FUNCTION_BLOCK TwoConRingCTL (* Composite Function Block Type *)
  (* Standard: 61499-2 *)
  (* Version 0.2, 2003-12-05, JHC, Rockwell Automation, Renamed from NEWCOMPFB. *)
  (* Version 0.1, 2002-01-08, JHC, Rockwell Automation, Added DLY FB as example. *)
  (* Version 0.0, 2000-05-27, JHC, Rockwell Automation *)
  (* Compiler header: package fb.rt.cs725; *)
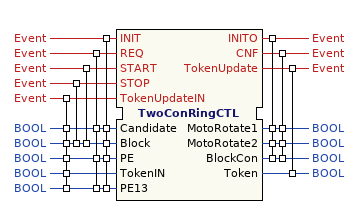
  EVENT_INPUT
    INIT WITH Candidate, Block, PE, PE13; (* Initialization Request *)
    REQ WITH Candidate, PE, PE13; (* Normal Execution Request *)
    START WITH Block;
    STOP WITH Block;
    TokenUpdateIN WITH Candidate, Block, PE, TokenIN, PE13;
  END_EVENT
  EVENT_OUTPUT
    INITO WITH MotoRotate1, MotoRotate2, BlockCon; (* Initialization Confirm *)
    CNF WITH MotoRotate1, MotoRotate2, BlockCon; (* Execution Confirmation *)
    TokenUpdate WITH Token;
  END_EVENT
  VAR_INPUT
    Candidate : BOOL;
    Block : BOOL;
    PE : BOOL;
    TokenIN : BOOL;
    PE13 : BOOL;
  END_VAR
  VAR_OUTPUT
    MotoRotate1 : BOOL;
    MotoRotate2 : BOOL;
    BlockCon : BOOL;
    Token : BOOL;
  END_VAR
  FBS
    FC11 : ConveyorCTL(PE := 0, Block := 0, Candidate := 0);
    Con4 : RingTokenHasCTL;
  END_FBS
  EVENT_CONNECTIONS
    INIT TO FC11.INIT;
    REQ TO FC11.REQ;
    Con4.INITO TO INITO;
    Con4.CNF TO CNF;
    REQ TO Con4.REQ;
    STOP TO Con4.CAS_STOP;
    START TO Con4.CAS_START;
    Con4.STOP TO FC11.CAS_STOP;
    Con4.START TO FC11.CAS_START;
    FC11.INITO TO Con4.INIT;
    Con4.TokenUpdate TO TokenUpdate;
    TokenUpdateIN TO Con4.TokenUpdateIN;
  END_CONNECTIONS
  DATA_CONNECTIONS
    Block TO Con4.Block;
    Candidate TO Con4.Candidate;
    PE TO Con4.PE;
    Con4.BlockCon TO BlockCon;
    FC11.MotoRotate TO MotoRotate1;
    Con4.MotoRotate TO MotoRotate2;
    PE13 TO Con4.PE13;
    TokenIN TO Con4.TokenIN;
    Con4.Token TO Token;
  END_CONNECTIONS
END_FUNCTION_BLOCK
